// LS Electric XG5000 project: onoffdelay
// PLC LSPLC
// module base 0 slot 0: 입출력 모듈:XBC-DR30S (DC 24V 입력 18점, 릴레이 출력 12점)

PROGRAM onoffdelay (task: 스캔 프로그램)

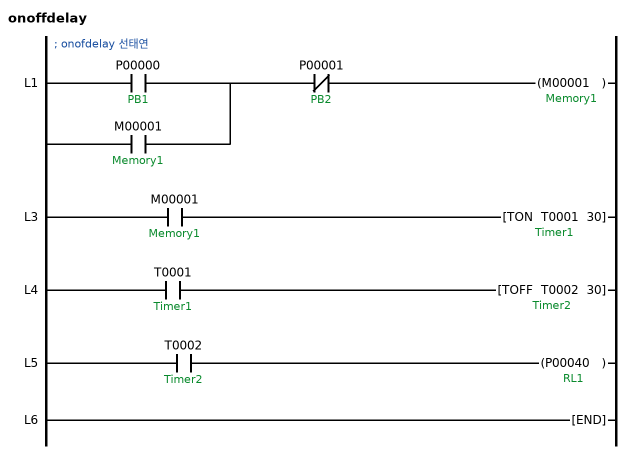
// onofdelay 선태연
; L1
LOAD      P00000	// PB1
OR        M00001	// Memory1
AND NOT   P00001	// PB2
OUT       M00001	// Memory1
; L3
LOAD      M00001	// Memory1
TON       T0001 30	// Timer1
; L4
LOAD      T0001	// Timer1
TOFF      T0002 30	// Timer2
; L5
LOAD      T0002	// Timer2
OUT       P00040	// RL1
; L6
END